TYPE ST_4PViciValveSampleNames :
STRUCT
      {attribute 'pytmc' := '
        pv: 01
        io: io
     '}
     s1 : STRING;
     {attribute 'pytmc' := '
        pv: 02
        io: io
     '}
     s2 : STRING;
     {attribute 'pytmc' := '
        pv: 03
        io: io
     '}
     s3 : STRING;
     {attribute 'pytmc' := '
        pv: 04
        io: io
     '}
     s4 : STRING;
END_STRUCT
END_TYPE

(* stored: Version 1.1.0.1, ProductVersion 3.1.4024.12
   DUT ST_4PViciValveSampleNames: Id {b42a57d8-e8a7-4340-891c-200ec30ff736} *)
